Staubli VAL3: getBoxSize.pgx

public program getBoxSize(num x_nType (dimensions=1), num& x_nSize (dimensions=1))
  local string l_sLibList
begin
  //得到所有回HOME设置数据文件库大小
  switch x_nType
    case 1
      //small box size
      x_nSize=size(sml:box)
    break
    case 2
      //big box size
      x_nSize=size(big:box)
    break
  endSwitch
end
